{attribute addProperty BoxType "EL6021-0000-0018"}
{attribute addProperty Id "COM_TxPDO_Map_InputsAT %I*COM_TxPDO_Map_Inputs_85D1D733192240COM_RxPDO_Map_OutputsAT %Q*COM_RxPDO_Map_Outputs_AC29F8FC192240WcStateAT %I*WcState_98A4DF7520.250InfoDataAT %I*InfoData_BC63D37F80100"}
{attribute addProperty CRC "620318934"}
{attribute addProperty SizeInBites "466"}
{attribute addProperty SizeInBytes "58.25"}
TYPE EL6021_8A84BDBB :
STRUCT
	{attribute addProperty Name "COM_TxPDO_Map_Inputs"}
	COM_TxPDO_Map_Inputs : COM_TxPDO_Map_Inputs_85D1D733;
	{attribute addProperty Name "COM_RxPDO_Map_Outputs"}
	COM_RxPDO_Map_Outputs : COM_RxPDO_Map_Outputs_AC29F8FC;
	{attribute addProperty Name "WcState"}
	WcState : WcState_98A4DF75;
	{attribute addProperty Name "InfoData"}
	InfoData : InfoData_BC63D37F;
END_STRUCT
END_TYPE

(* stored: Version 1.2.0.0, ProductVersion 3.1.4024.9
   DUT EL6021_8A84BDBB: Id {d0447e71-358d-47d9-bfbe-8ea7f5fe0b75} *)
